PROGRAM PRG_PLAS_11_PackAggregationCtrl
VAR
	tonEnableCameraSystem					: TON;
	bEnablePackTriggeringAfterDelay			: BOOL;
	bEnablePackAggregationCameraSystem	: BOOL;

	tofPackAggregationCameraOFFDelay 		: TOF;

	rsInhibitCameraTrigger				: RS;
	rtrigNewArrived						: R_TRIG;
	bNewCodeIsProccesing				: BOOL;

	fbCodeDiag							: FB_SCANNER_DiagnosticLog;

	tonValidationTimout					: TON;
	bValidationTimeout					: BOOL;
	bValidationTimeoutReset				: BOOL;

	fbPackAggregationCamera				: FB_SCANNER_CameraSelect;
	fbPackAggregationEvaluation			: FB_SCANNER_Evaluation;

	rtPackAggregationCameraDone		:  R_TRIG;
	bPackAggregationCameraDone		:  BOOL;

	fbAddPacksToInfeedQ					: FB_T03_AddMultiPackToInfeedQ;
	fbFillInPackInfeedQueue				: FB_PLAS_MasterListFillInPackRev;

	fbDebugCNT							: FB_DEBUG_CounterArray;
	aCNTDebug							: ARRAY [1..10] OF UDINT;
	bResetCNT								: BOOL;

END_VAR
VAR // added by the converter: edge detectors and wires of the graphical bodies
    _w1 : BOOL;
END_VAR

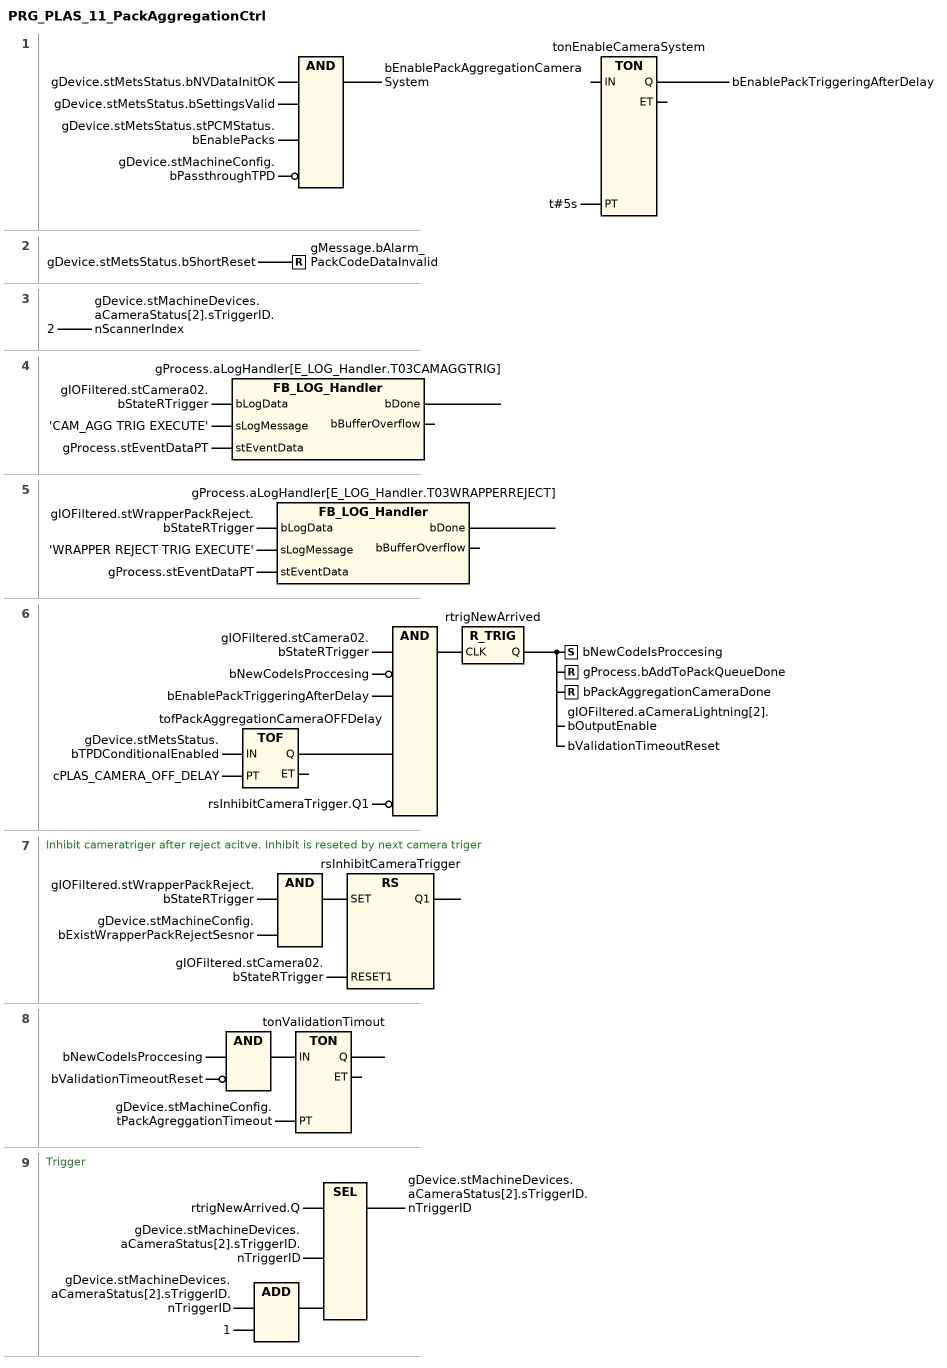
// NETWORK 1
_w1 := gDevice.stMetsStatus.bNVDataInitOK AND gDevice.stMetsStatus.bSettingsValid AND gDevice.stMetsStatus.stPCMStatus.bEnablePacks AND NOT gDevice.stMachineConfig.bPassthroughTPD;
bEnablePackAggregationCameraSystem := _w1;
tonEnableCameraSystem(IN := _w1, PT := t#5s); // TON
bEnablePackTriggeringAfterDelay := tonEnableCameraSystem.Q;

// NETWORK 2
gMessage.bAlarm_PackCodeDataInvalid R= gDevice.stMetsStatus.bShortReset;

// NETWORK 3
gDevice.stMachineDevices.aCameraStatus[2].sTriggerID.nScannerIndex := 2;

// NETWORK 4
gProcess.aLogHandler[E_LOG_Handler.T03CAMAGGTRIG](
    bLogData := gIOFiltered.stCamera02.bStateRTrigger,
    sLogMessage := 'CAM_AGG TRIG EXECUTE',
    stEventData := gProcess.stEventDataPT); // FB_LOG_Handler

// NETWORK 5
gProcess.aLogHandler[E_LOG_Handler.T03WRAPPERREJECT](
    bLogData := gIOFiltered.stWrapperPackReject.bStateRTrigger,
    sLogMessage := 'WRAPPER REJECT TRIG EXECUTE',
    stEventData := gProcess.stEventDataPT); // FB_LOG_Handler

// NETWORK 6
tofPackAggregationCameraOFFDelay(IN := gDevice.stMetsStatus.bTPDConditionalEnabled, PT := cPLAS_CAMERA_OFF_DELAY); // TOF
rtrigNewArrived(CLK := gIOFiltered.stCamera02.bStateRTrigger AND NOT bNewCodeIsProccesing AND bEnablePackTriggeringAfterDelay AND tofPackAggregationCameraOFFDelay.Q AND NOT rsInhibitCameraTrigger.Q1); // R_TRIG
bNewCodeIsProccesing S= rtrigNewArrived.Q;
gProcess.bAddToPackQueueDone R= rtrigNewArrived.Q;
bPackAggregationCameraDone R= rtrigNewArrived.Q;
gIOFiltered.aCameraLightning[2].bOutputEnable := rtrigNewArrived.Q;
bValidationTimeoutReset := rtrigNewArrived.Q;

// NETWORK 7
// Inhibit cameratriger after reject acitve. Inhibit is reseted by next camera triger
rsInhibitCameraTrigger(SET := gIOFiltered.stWrapperPackReject.bStateRTrigger AND gDevice.stMachineConfig.bExistWrapperPackRejectSesnor, RESET1 := gIOFiltered.stCamera02.bStateRTrigger); // RS

// NETWORK 8
tonValidationTimout(IN := bNewCodeIsProccesing AND NOT bValidationTimeoutReset, PT := gDevice.stMachineConfig.tPackAgreggationTimeout); // TON

// NETWORK 9
// Trigger
gDevice.stMachineDevices.aCameraStatus[2].sTriggerID.nTriggerID := SEL(rtrigNewArrived.Q, gDevice.stMachineDevices.aCameraStatus[2].sTriggerID.nTriggerID, gDevice.stMachineDevices.aCameraStatus[2].sTriggerID.nTriggerID + 1);

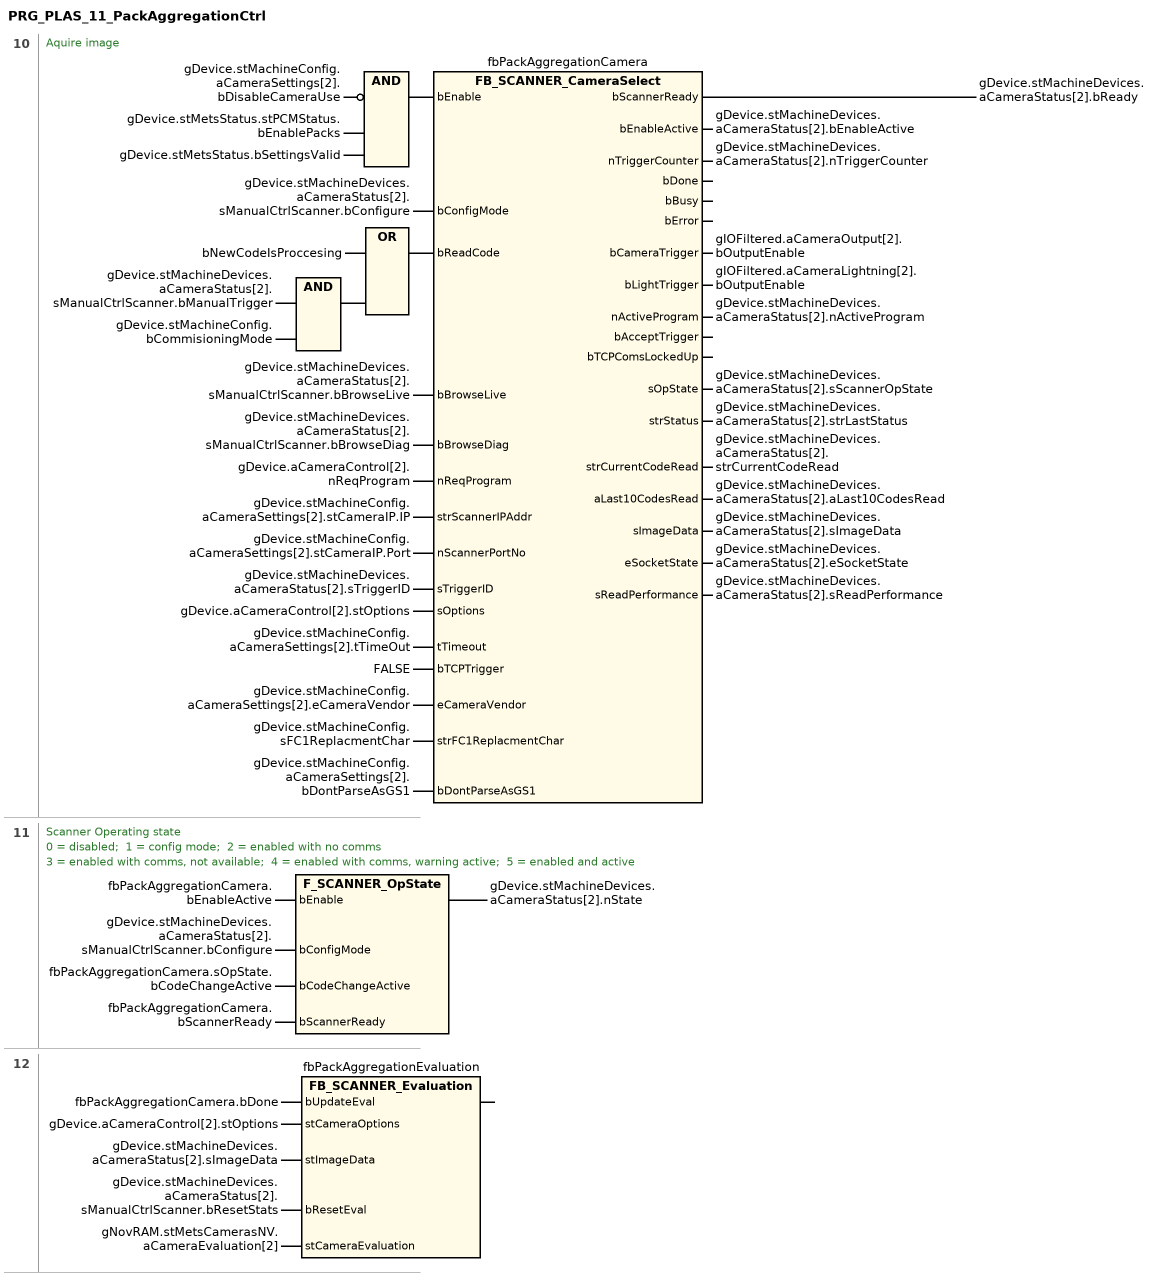
// NETWORK 10
// Aquire image
fbPackAggregationCamera(
    bEnable := NOT gDevice.stMachineConfig.aCameraSettings[2].bDisableCameraUse AND gDevice.stMetsStatus.stPCMStatus.bEnablePacks AND gDevice.stMetsStatus.bSettingsValid,
    bConfigMode := gDevice.stMachineDevices.aCameraStatus[2].sManualCtrlScanner.bConfigure,
    bReadCode := bNewCodeIsProccesing OR gDevice.stMachineDevices.aCameraStatus[2].sManualCtrlScanner.bManualTrigger AND gDevice.stMachineConfig.bCommisioningMode,
    bBrowseLive := gDevice.stMachineDevices.aCameraStatus[2].sManualCtrlScanner.bBrowseLive,
    bBrowseDiag := gDevice.stMachineDevices.aCameraStatus[2].sManualCtrlScanner.bBrowseDiag,
    nReqProgram := gDevice.aCameraControl[2].nReqProgram,
    strScannerIPAddr := gDevice.stMachineConfig.aCameraSettings[2].stCameraIP.IP,
    nScannerPortNo := gDevice.stMachineConfig.aCameraSettings[2].stCameraIP.Port,
    sTriggerID := gDevice.stMachineDevices.aCameraStatus[2].sTriggerID,
    sOptions := gDevice.aCameraControl[2].stOptions,
    tTimeout := gDevice.stMachineConfig.aCameraSettings[2].tTimeOut,
    bTCPTrigger := FALSE,
    eCameraVendor := gDevice.stMachineConfig.aCameraSettings[2].eCameraVendor,
    strFC1ReplacmentChar := gDevice.stMachineConfig.sFC1ReplacmentChar,
    bDontParseAsGS1 := gDevice.stMachineConfig.aCameraSettings[2].bDontParseAsGS1,
    bEnableActive => gDevice.stMachineDevices.aCameraStatus[2].bEnableActive,
    nTriggerCounter => gDevice.stMachineDevices.aCameraStatus[2].nTriggerCounter,
    bCameraTrigger => gIOFiltered.aCameraOutput[2].bOutputEnable,
    bLightTrigger => gIOFiltered.aCameraLightning[2].bOutputEnable,
    nActiveProgram => gDevice.stMachineDevices.aCameraStatus[2].nActiveProgram,
    sOpState => gDevice.stMachineDevices.aCameraStatus[2].sScannerOpState,
    strStatus => gDevice.stMachineDevices.aCameraStatus[2].strLastStatus,
    strCurrentCodeRead => gDevice.stMachineDevices.aCameraStatus[2].strCurrentCodeRead,
    aLast10CodesRead => gDevice.stMachineDevices.aCameraStatus[2].aLast10CodesRead,
    sImageData => gDevice.stMachineDevices.aCameraStatus[2].sImageData,
    eSocketState => gDevice.stMachineDevices.aCameraStatus[2].eSocketState,
    sReadPerformance => gDevice.stMachineDevices.aCameraStatus[2].sReadPerformance); // FB_SCANNER_CameraSelect
gDevice.stMachineDevices.aCameraStatus[2].bReady := fbPackAggregationCamera.bScannerReady;

// NETWORK 11
// 					Scanner Operating state
// 0 = disabled;  1 = config mode;  2 = enabled with no comms
// 3 = enabled with comms, not available;  4 = enabled with comms, warning active;  5 = enabled and active
//
gDevice.stMachineDevices.aCameraStatus[2].nState := F_SCANNER_OpState(bEnable := fbPackAggregationCamera.bEnableActive, bConfigMode := gDevice.stMachineDevices.aCameraStatus[2].sManualCtrlScanner.bConfigure, bCodeChangeActive := fbPackAggregationCamera.sOpState.bCodeChangeActive, bScannerReady := fbPackAggregationCamera.bScannerReady);

// NETWORK 12
fbPackAggregationEvaluation(
    bUpdateEval := fbPackAggregationCamera.bDone,
    stCameraOptions := gDevice.aCameraControl[2].stOptions,
    stImageData := gDevice.stMachineDevices.aCameraStatus[2].sImageData,
    bResetEval := gDevice.stMachineDevices.aCameraStatus[2].sManualCtrlScanner.bResetStats,
    stCameraEvaluation := gNovRAM.stMetsCamerasNV.aCameraEvaluation[2]); // FB_SCANNER_Evaluation

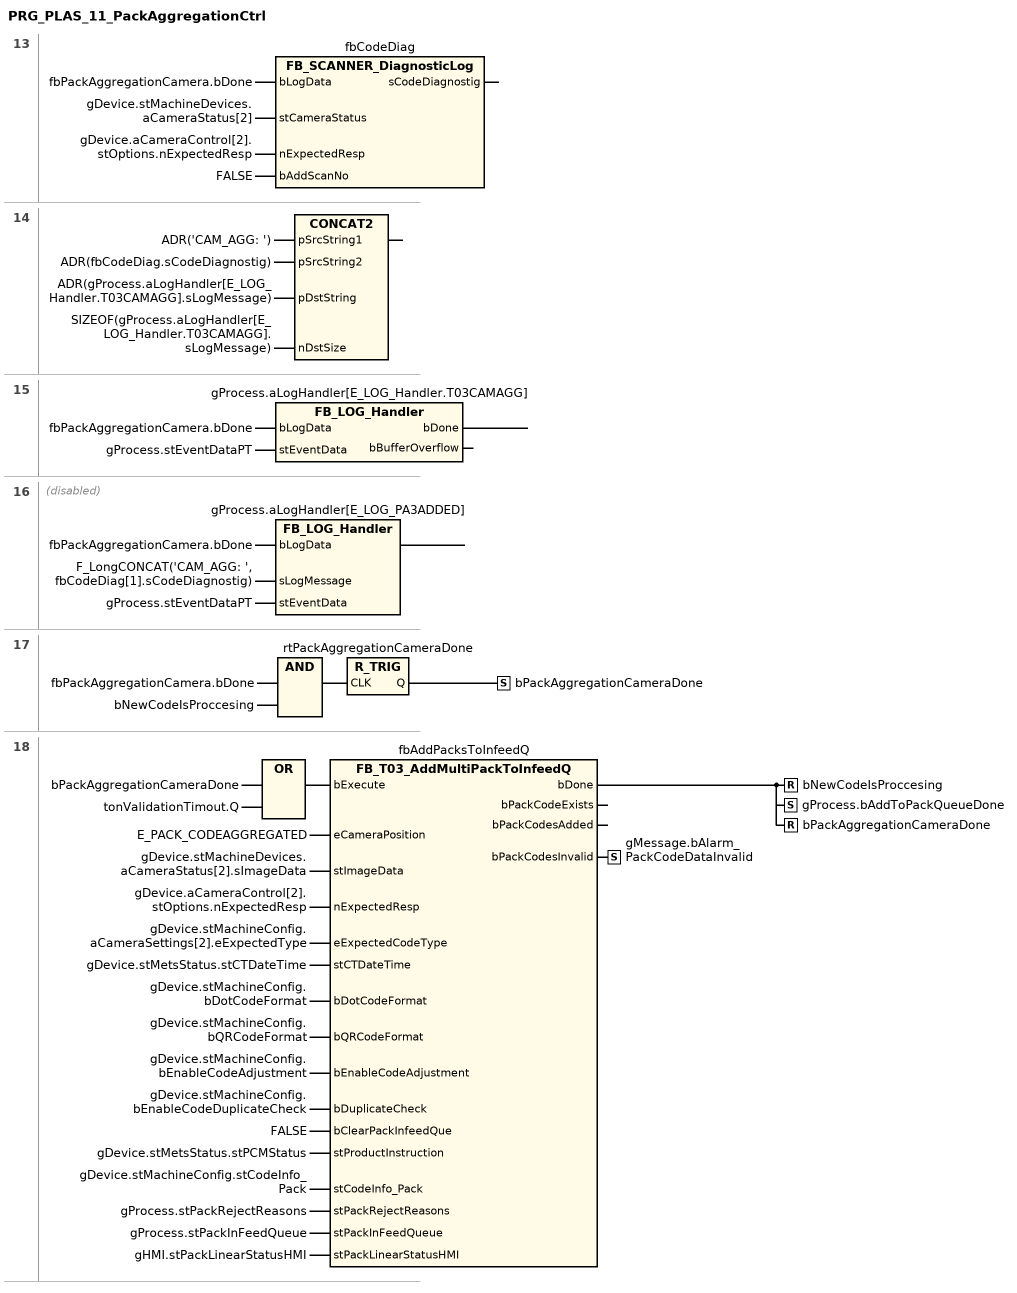
// NETWORK 13
fbCodeDiag(
    bLogData := fbPackAggregationCamera.bDone,
    stCameraStatus := gDevice.stMachineDevices.aCameraStatus[2],
    nExpectedResp := gDevice.aCameraControl[2].stOptions.nExpectedResp,
    bAddScanNo := FALSE); // FB_SCANNER_DiagnosticLog

// NETWORK 14
CONCAT2(pSrcString1 := ADR('CAM_AGG: '), pSrcString2 := ADR(fbCodeDiag.sCodeDiagnostig), pDstString := ADR(gProcess.aLogHandler[E_LOG_Handler.T03CAMAGG].sLogMessage), nDstSize := SIZEOF(gProcess.aLogHandler[E_LOG_Handler.T03CAMAGG].sLogMessage));

// NETWORK 15
gProcess.aLogHandler[E_LOG_Handler.T03CAMAGG](bLogData := fbPackAggregationCamera.bDone, stEventData := gProcess.stEventDataPT); // FB_LOG_Handler

// NETWORK 16 (disabled)
// gProcess.aLogHandler[E_LOG_PA3ADDED](
//     bLogData := fbPackAggregationCamera.bDone,
//     sLogMessage := F_LongCONCAT('CAM_AGG: ', fbCodeDiag[1].sCodeDiagnostig),
//     stEventData := gProcess.stEventDataPT); // FB_LOG_Handler

// NETWORK 17
rtPackAggregationCameraDone(CLK := fbPackAggregationCamera.bDone AND bNewCodeIsProccesing); // R_TRIG
bPackAggregationCameraDone S= rtPackAggregationCameraDone.Q;

// NETWORK 18
fbAddPacksToInfeedQ(
    bExecute := bPackAggregationCameraDone OR tonValidationTimout.Q,
    eCameraPosition := E_PACK_CODEAGGREGATED,
    stImageData := gDevice.stMachineDevices.aCameraStatus[2].sImageData,
    nExpectedResp := gDevice.aCameraControl[2].stOptions.nExpectedResp,
    eExpectedCodeType := gDevice.stMachineConfig.aCameraSettings[2].eExpectedType,
    stCTDateTime := gDevice.stMetsStatus.stCTDateTime,
    bDotCodeFormat := gDevice.stMachineConfig.bDotCodeFormat,
    bQRCodeFormat := gDevice.stMachineConfig.bQRCodeFormat,
    bEnableCodeAdjustment := gDevice.stMachineConfig.bEnableCodeAdjustment,
    bDuplicateCheck := gDevice.stMachineConfig.bEnableCodeDuplicateCheck,
    bClearPackInfeedQue := FALSE,
    stProductInstruction := gDevice.stMetsStatus.stPCMStatus,
    stCodeInfo_Pack := gDevice.stMachineConfig.stCodeInfo_Pack,
    stPackRejectReasons := gProcess.stPackRejectReasons,
    stPackInFeedQueue := gProcess.stPackInFeedQueue,
    stPackLinearStatusHMI := gHMI.stPackLinearStatusHMI); // FB_T03_AddMultiPackToInfeedQ
gMessage.bAlarm_PackCodeDataInvalid S= fbAddPacksToInfeedQ.bPackCodesInvalid;
bNewCodeIsProccesing R= fbAddPacksToInfeedQ.bDone;
gProcess.bAddToPackQueueDone S= fbAddPacksToInfeedQ.bDone;
bPackAggregationCameraDone R= fbAddPacksToInfeedQ.bDone;

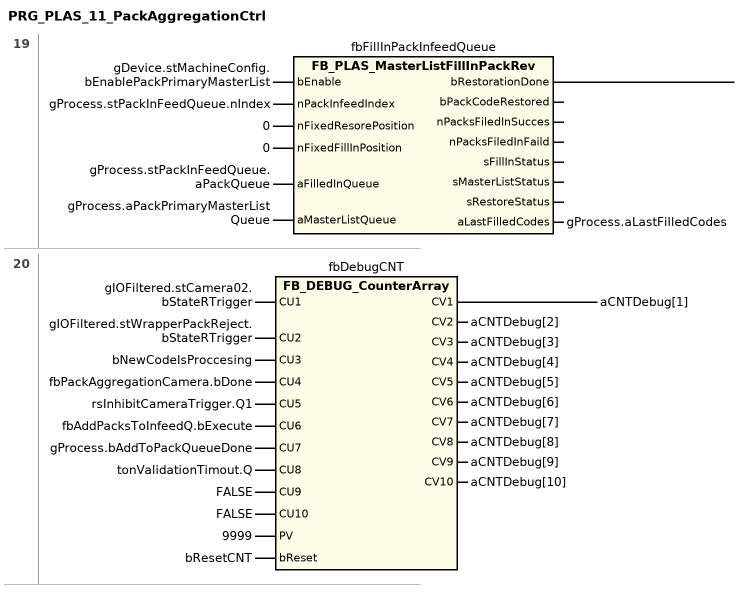
// NETWORK 19
fbFillInPackInfeedQueue(
    bEnable := gDevice.stMachineConfig.bEnablePackPrimaryMasterList,
    nPackInfeedIndex := gProcess.stPackInFeedQueue.nIndex,
    nFixedResorePosition := 0,
    nFixedFillInPosition := 0,
    aFilledInQueue := gProcess.stPackInFeedQueue.aPackQueue,
    aMasterListQueue := gProcess.aPackPrimaryMasterListQueue,
    aLastFilledCodes => gProcess.aLastFilledCodes); // FB_PLAS_MasterListFillInPackRev

// NETWORK 20
fbDebugCNT(
    CU1 := gIOFiltered.stCamera02.bStateRTrigger,
    CU2 := gIOFiltered.stWrapperPackReject.bStateRTrigger,
    CU3 := bNewCodeIsProccesing,
    CU4 := fbPackAggregationCamera.bDone,
    CU5 := rsInhibitCameraTrigger.Q1,
    CU6 := fbAddPacksToInfeedQ.bExecute,
    CU7 := gProcess.bAddToPackQueueDone,
    CU8 := tonValidationTimout.Q,
    CU9 := FALSE,
    CU10 := FALSE,
    PV := 9999,
    bReset := bResetCNT,
    CV2 => aCNTDebug[2],
    CV3 => aCNTDebug[3],
    CV4 => aCNTDebug[4],
    CV5 => aCNTDebug[5],
    CV6 => aCNTDebug[6],
    CV7 => aCNTDebug[7],
    CV8 => aCNTDebug[8],
    CV9 => aCNTDebug[9],
    CV10 => aCNTDebug[10]); // FB_DEBUG_CounterArray
aCNTDebug[1] := fbDebugCNT.CV1;

END_PROGRAM

(* stored: Version 1.1.0.1
   POU PRG_PLAS_11_PackAggregationCtrl: Id {8ee3d69b-6b4a-4978-b032-85c733d51d84}, SpecialFunc None *)
